# EPICS StreamDevice protocol: ESP8266/proto/bme280.proto
OutTerminator = LF;

getTemp{
	out "getTemperature";
	in "%f";
}

getHumi{
	out "getHumidity";
	in "%f";
}

getPres{
	out "getPressure";
	in "%f";
}
